Staubli VAL3: onEnterEvent.pgx

program onEnterEvent()
  local num l_nResult
  local string l_sMessage
  local string l_sMessage2
  local string l_sMessage3
  local string l_sItem
begin
  //if saveData:mode>0
  if !bPage
    //
    //  open the processes list PAGE
    //
    //      saveData:sProcessList="default"
    //      call processList:loadProcessList(saveData:sProcessList,l_nResult)
    l_sItem="true"
    call loadPage("kernel/page/processList",l_sItem)
    // came back
    logMsg("[KERNEL] INTERFACE:PAGE Production")
    // refresh
    cls()
    use:bUseRefresh=true
  endIf
  //endIf
end
